FUNCTION_BLOCK Physical_Plant_SIMULATION (* Composite Function Block Type *)
  (* Standard: 61499-2 *)
  (* Version 0.0, 12/12/2023, Cheyan, Schneider Electric, template *)
  PACKAGE Main;
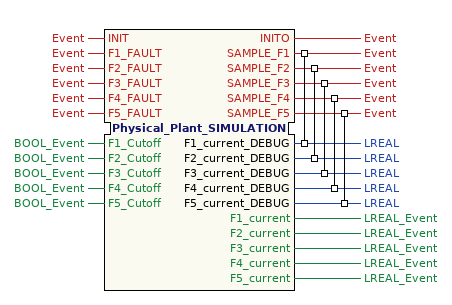
  EVENT_INPUT
    INIT; (* Initialization Request *)
    F1_FAULT;
    F2_FAULT;
    F3_FAULT;
    F4_FAULT;
    F5_FAULT;
  END_EVENT
  EVENT_OUTPUT
    INITO; (* Initialization Confirm *)
    SAMPLE_F1 WITH F1_current_DEBUG;
    SAMPLE_F2 WITH F2_current_DEBUG;
    SAMPLE_F3 WITH F3_current_DEBUG;
    SAMPLE_F4 WITH F4_current_DEBUG;
    SAMPLE_F5 WITH F5_current_DEBUG;
  END_EVENT
  VAR_OUTPUT
    F1_current_DEBUG : LREAL; (* Output event qualifier *)
    F2_current_DEBUG : LREAL; (* Output event qualifier *)
    F3_current_DEBUG : LREAL; (* Output event qualifier *)
    F4_current_DEBUG : LREAL; (* Output event qualifier *)
    F5_current_DEBUG : LREAL; (* Output event qualifier *)
  END_VAR
  SOCKETS
    F1_Cutoff : BOOL_Event;
    F2_Cutoff : BOOL_Event;
    F3_Cutoff : BOOL_Event;
    F4_Cutoff : BOOL_Event;
    F5_Cutoff : BOOL_Event;
  END_SOCKETS
  PLUGS
    F1_current : LREAL_Event;
    F2_current : LREAL_Event;
    F3_current : LREAL_Event;
    F4_current : LREAL_Event;
    F5_current : LREAL_Event;
  END_PLUGS
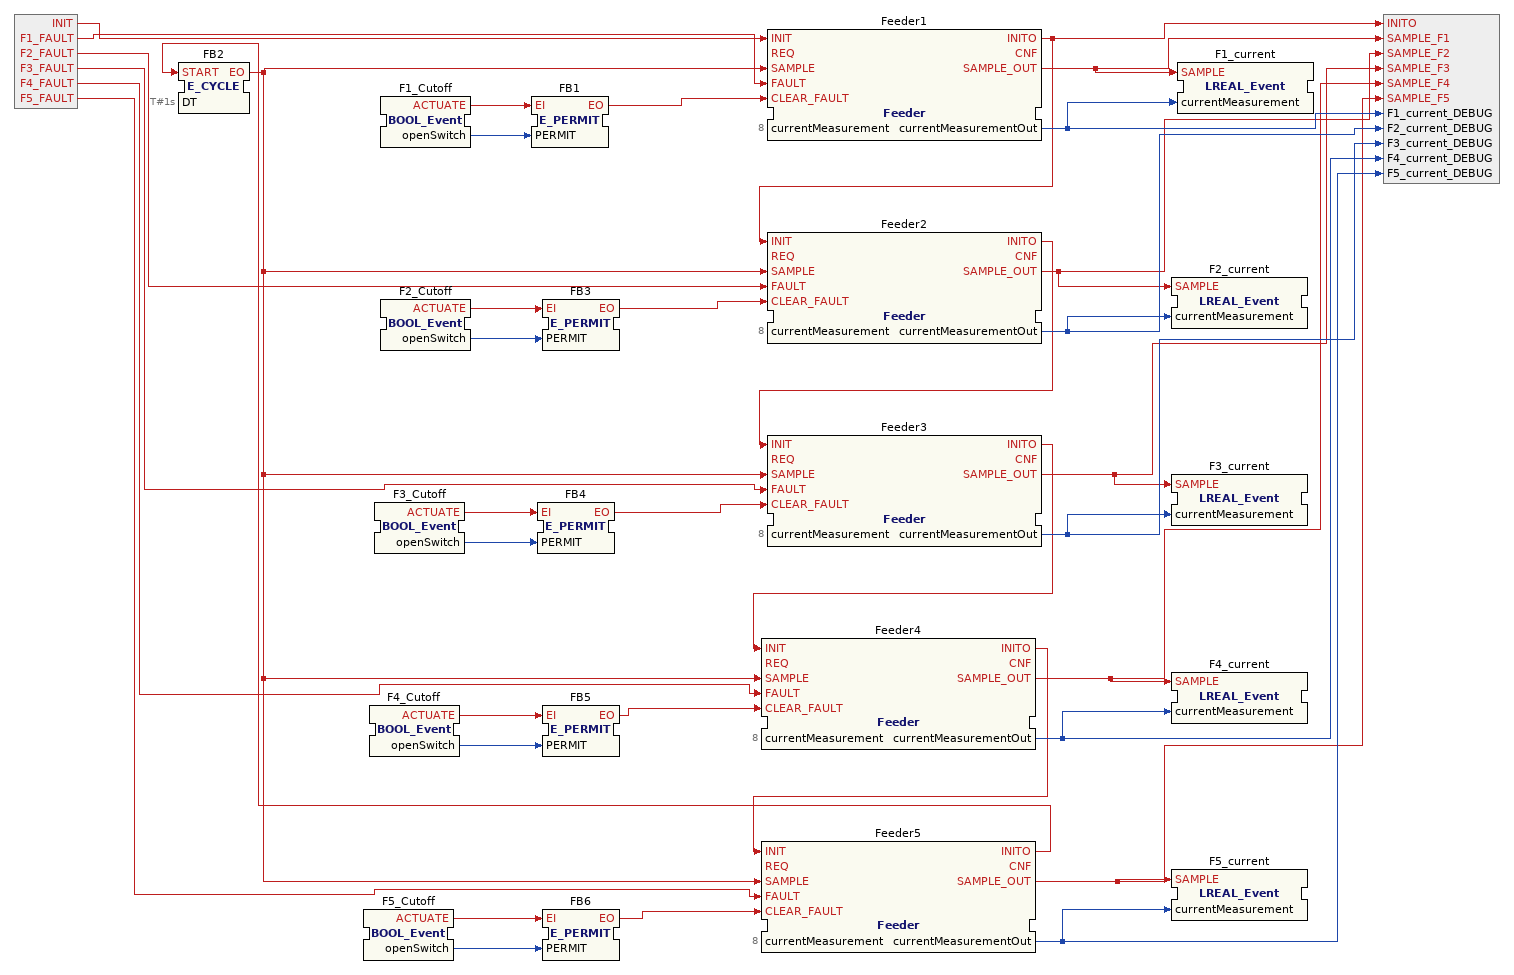
  FBS
    Feeder1 : Feeder(currentMeasurement := 8);
    FB2 : E_CYCLE(DT := T#1s);
    Feeder2 : Feeder(currentMeasurement := 8);
    Feeder3 : Feeder(currentMeasurement := 8);
    Feeder4 : Feeder(currentMeasurement := 8);
    Feeder5 : Feeder(currentMeasurement := 8);
    FB1 : E_PERMIT;
    FB3 : E_PERMIT;
    FB4 : E_PERMIT;
    FB5 : E_PERMIT;
    FB6 : E_PERMIT;
  END_FBS
  EVENT_CONNECTIONS
    FB2.EO TO Feeder1.SAMPLE;
    INIT TO Feeder1.INIT;
    Feeder1.INITO TO Feeder2.INIT;
    Feeder2.INITO TO Feeder3.INIT;
    Feeder3.INITO TO Feeder4.INIT;
    Feeder4.INITO TO Feeder5.INIT;
    Feeder5.INITO TO FB2.START;
    F1_FAULT TO Feeder1.FAULT;
    F2_FAULT TO Feeder2.FAULT;
    FB2.EO TO Feeder2.SAMPLE;
    FB2.EO TO Feeder3.SAMPLE;
    F3_FAULT TO Feeder3.FAULT;
    F4_FAULT TO Feeder4.FAULT;
    FB2.EO TO Feeder4.SAMPLE;
    FB2.EO TO Feeder5.SAMPLE;
    F5_FAULT TO Feeder5.FAULT;
    Feeder1.SAMPLE_OUT TO SAMPLE_F1;
    Feeder1.INITO TO INITO;
    Feeder2.SAMPLE_OUT TO SAMPLE_F2;
    Feeder3.SAMPLE_OUT TO SAMPLE_F3;
    Feeder4.SAMPLE_OUT TO SAMPLE_F4;
    Feeder5.SAMPLE_OUT TO SAMPLE_F5;
    Feeder1.SAMPLE_OUT TO F1_current.SAMPLE;
    Feeder2.SAMPLE_OUT TO F2_current.SAMPLE;
    Feeder3.SAMPLE_OUT TO F3_current.SAMPLE;
    Feeder4.SAMPLE_OUT TO F4_current.SAMPLE;
    Feeder5.SAMPLE_OUT TO F5_current.SAMPLE;
    F1_Cutoff.ACTUATE TO FB1.EI;
    FB1.EO TO Feeder1.CLEAR_FAULT;
    F2_Cutoff.ACTUATE TO FB3.EI;
    FB3.EO TO Feeder2.CLEAR_FAULT;
    F3_Cutoff.ACTUATE TO FB4.EI;
    FB4.EO TO Feeder3.CLEAR_FAULT;
    F4_Cutoff.ACTUATE TO FB5.EI;
    FB5.EO TO Feeder4.CLEAR_FAULT;
    F5_Cutoff.ACTUATE TO FB6.EI;
    FB6.EO TO Feeder5.CLEAR_FAULT;
  END_CONNECTIONS
  DATA_CONNECTIONS
    Feeder1.currentMeasurementOut TO F1_current_DEBUG;
    Feeder2.currentMeasurementOut TO F2_current_DEBUG;
    Feeder3.currentMeasurementOut TO F3_current_DEBUG;
    Feeder4.currentMeasurementOut TO F4_current_DEBUG;
    Feeder5.currentMeasurementOut TO F5_current_DEBUG;
    Feeder1.currentMeasurementOut TO F1_current.currentMeasurement;
    Feeder2.currentMeasurementOut TO F2_current.currentMeasurement;
    Feeder3.currentMeasurementOut TO F3_current.currentMeasurement;
    Feeder4.currentMeasurementOut TO F4_current.currentMeasurement;
    Feeder5.currentMeasurementOut TO F5_current.currentMeasurement;
    F1_Cutoff.openSwitch TO FB1.PERMIT;
    F2_Cutoff.openSwitch TO FB3.PERMIT;
    F3_Cutoff.openSwitch TO FB4.PERMIT;
    F4_Cutoff.openSwitch TO FB5.PERMIT;
    F5_Cutoff.openSwitch TO FB6.PERMIT;
  END_CONNECTIONS
END_FUNCTION_BLOCK
